Staubli VAL3: moveY.pgx

public program moveY(num nDy (dimensions=1))
  local point pFinal
  local point pHere
begin
  //pHere=here(tActive,frActive)
  //pFinal=compose(pHere,frActive,{0,nDy,0,0,0,0})
  //movel(pFinal,tActive,mNomSpeed)
  pDest=compose(pDest,frActive,{0,nDy,0,0,0,0})
  movel(pDest,tActive,mNomSpeed)
end
